// TwinCAT 3 PLC project Bsc_NoComp
// ProgramVersion: 3.1.4024.0
// libraries:
//   CmpBitmapPool, * (System)
//   Tc2_Standard, * (Beckhoff Automation GmbH)
//   Tc2_System, * (Beckhoff Automation GmbH)
//   Tc3_Module, * (Beckhoff Automation GmbH)
//   VisuSymbols,3.5.10.0,System
// project tree:
//   / GlobalTextList.TcGTLO (not stored), PlcTask.TcTTO, Visualization Manager.TcVMO (not stored)
//   GVLs/ G_Enables.TcGVL (not stored), G_FilterConstants.TcGVL (not stored), G_Mode.TcGVL, G_OPC.TcGVL (not stored), G_Parameters.TcGVL (not stored)
//   Input/ G_Input.TcGVL (not stored)
//   Output/ G_Output.TcGVL (not stored)
//   Program/ MAIN.TcPOU (not stored)
//   XML/ FB_Derivator.TcPOU (not stored), FB_Integrator.TcPOU (not stored), G_Init.TcGVL (not stored)

CONFIGURATION Bsc_NoComp
    RESOURCE PLC ON TwinCAT3
        TASK PlcTask(INTERVAL := T#1ms, PRIORITY := 20);
        PROGRAM MAIN WITH PlcTask : MAIN;
    END_RESOURCE
END_CONFIGURATION

// ---- GVLs/G_Mode.TcGVL
{attribute 'qualified_only'}
VAR_GLOBAL
END_VAR
